Yaskawa INFORM job: R1_W29-KM-NOWY-MP.JBI

/JOB
//NAME R1_W29-KM-NOWY-MP
///FOLDERNAME KRIS-SCIANA
//POS
///NPOS 90,90,76,8,0,0
///TOOL 0
///POSTYPE PULSE
///PULSE
C00000=-43238,-20123,-76298,22793,79190,-61716
C00001=-147206,-71099,-63807,5032,65627,-10001
C00002=-131466,-57276,-50947,-729,64392,-4195
C00003=-131466,-55755,-45239,-747,61662,-4178
C00004=-113506,-33937,-32252,-19801,72986,17092
C00005=-113506,-33758,-31414,-19844,72586,17160
C00006=-113506,-33937,-32252,-19801,72986,17092
C00007=-112868,-36448,-33885,-19979,72871,17349
C00008=-112868,-36201,-32777,-20033,72350,17439
C00009=-113561,-35138,-32088,-19860,72296,17187
C00010=-112868,-36340,-33394,-20002,72641,17389
C00011=-112868,-36673,-34952,-19926,73383,17263
C00012=-136354,-51968,-44201,-1495,62997,-3424
C00013=-136354,-51734,-43329,-1501,62580,-3419
C00014=-136354,-51441,-42272,-1507,62080,-3413
C00015=-136354,-51646,-43010,-1502,62428,-3418
C00016=-136803,-55259,-45028,-1340,61807,-3581
C00017=-136803,-54973,-44058,-1346,61359,-3576
C00018=-136592,-53313,-43138,-1422,61645,-3500
C00019=-136869,-55877,-45678,-1314,61887,-3609
C00020=-144453,-49639,-42868,1535,63375,-6471
C00021=-144614,-48538,-41583,1597,63154,-6534
C00022=-144614,-48258,-40519,1602,62642,-6539
C00023=-144614,-48586,-41775,1593,63247,-6530
C00024=-145217,-51775,-43610,1827,62750,-6765
C00025=-145217,-51364,-42122,1839,62044,-6776
C00026=-144853,-49477,-41036,1695,62343,-6629
C00027=-145217,-51972,-44358,1823,63105,-6759
C00028=-157952,-18054,-25591,12162,79581,-30610
C00029=-158728,-15189,-23240,12317,79720,-30867
C00030=-158728,-15023,-21819,12345,78948,-30943
C00031=-158728,-15162,-22988,12322,79583,-30880
C00032=-160150,-16225,-23788,12608,79748,-31358
C00033=-160150,-16053,-22382,12636,78987,-31435
C00034=-159415,-15465,-21940,12489,78902,-31189
C00035=-160223,-15954,-23704,12620,79843,-31375
C00036=-161879,-22316,-38337,12820,85699,-31343
C00037=-142488,6647,-16194,-2372,99815,22094
C00038=-133363,46346,29890,-18296,105117,75189
C00039=-134257,47901,36105,-18159,102036,75336
C00040=-135288,44692,32242,-18369,102497,74886
C00041=-135288,44939,33433,-18321,101921,74975
C00042=-135288,44745,32503,-18359,102370,74905
C00043=-135129,47566,35532,-18302,102012,75019
C00044=-134852,48227,37162,-18209,101441,75210
C00045=-135455,46185,34960,-18323,101598,74964
C00046=-134852,48227,37162,-18209,101441,75210
C00047=-127142,35074,22200,-17190,105451,77446
C00048=-127142,35126,22513,-17174,105291,77468
C00049=-127142,35298,23490,-17124,104803,77542
C00050=-127142,35126,22513,-17174,105291,77468
C00051=-126238,38948,26146,-16993,105220,77814
C00052=-125881,39159,27623,-16857,104529,78046
C00053=-125732,37116,25510,-16853,104799,78062
C00054=-125881,39159,27623,-16857,104529,78046
C00055=-118491,39693,25202,-15641,107701,80341
C00056=-118491,40027,27191,-15541,106685,80478
C00057=-118491,40312,28701,-15455,105931,80575
C00058=-118491,40115,27679,-15502,106441,80508
C00059=-118523,43718,31472,-15465,105969,80559
C00060=-118523,43964,32657,-15412,105387,80635
C00061=-118326,41786,30355,-15400,105712,80665
C00062=-118523,43964,32657,-15412,105387,80635
C00063=-118101,6095,-16714,-15495,98189,81670
C00064=-121393,-29377,-38195,-9470,79556,5065
C00065=-135587,-47759,-49879,-6114,75955,393
C00066=-135563,-42241,-39607,-6218,72490,575
C00067=-148370,-35238,-35185,1969,72538,-10310
C00068=-156952,-26882,-29550,12128,77113,-24719
C00069=-159766,-12416,-18981,12668,78449,-25578
C00070=-155246,-26379,-37143,3868,78146,-24514
C00071=-111750,-20922,-29619,-16910,84852,24161
C00072=-112985,-19212,-23920,-16796,82079,24108
C00073=-118831,-30060,-31314,-15936,79920,22326
C00074=-124977,-39388,-37559,-9656,73919,11756
C00075=-135123,-42820,-39976,-5392,72032,5771
C00076=-141350,-43617,-40361,1374,71221,-3156
C00077=-141351,-45056,-47095,1351,74625,-3115
C00078=-142962,-17809,-31450,1751,79026,-53612
C00079=-136048,25460,5355,-7693,98061,-70296
C00080=-129481,56377,46609,-18750,110732,-89791
C00081=-130454,29429,16363,-16121,101280,-88696
C00082=-134058,37349,27654,-26404,95753,-89965
C00083=-134055,36228,21042,-26664,98897,-90683
C00084=-119345,38761,21089,-14797,104992,-85146
C00085=-121095,38621,26360,-13285,104325,-87017
C00086=-134151,52750,43450,-11485,107873,-85219
C00087=-130248,33721,13027,-16263,105211,-80194
C00088=-133531,-22452,-45998,-16065,102330,-23096
C00089=-43238,-20123,-76298,22793,79190,-61716
BC00000=125007,760961,1070891
BC00001=266312,761507,1070908
BC00002=266312,761507,1070908
BC00003=266312,761507,1070908
BC00004=266312,761507,1070908
BC00005=266312,761507,1070908
BC00006=266312,761507,1070908
BC00007=266312,761507,1070908
BC00008=266312,761507,1070908
BC00009=266312,761507,1070908
BC00010=266312,761507,1070908
BC00011=266312,761507,1070908
BC00012=266312,761507,1070908
BC00013=266312,761507,1070908
BC00014=266312,761507,1070908
BC00015=266312,761507,1070908
BC00016=266312,761507,1070908
BC00017=266312,761507,1070908
BC00018=266312,761507,1070908
BC00019=266312,761507,1070908
BC00020=266312,761507,1070908
BC00021=266312,761507,1070908
BC00022=266312,761507,1070908
BC00023=266312,761507,1070908
BC00024=266312,761507,1070908
BC00025=266312,761507,1070908
BC00026=266312,761507,1070908
BC00027=266312,761507,1070908
BC00028=266312,761507,1070908
BC00029=266312,761507,1070908
BC00030=266312,761507,1070908
BC00031=266312,761507,1070908
BC00032=266312,761507,1070908
BC00033=266312,761507,1070908
BC00034=266312,761507,1070908
BC00035=266312,761507,1070908
BC00036=266312,761507,1070908
BC00037=266312,761507,1070908
BC00038=266312,761507,1070908
BC00039=266312,761507,1070908
BC00040=266312,761507,1070908
BC00041=266312,761507,1070908
BC00042=266312,761507,1070908
BC00043=266312,761507,1070908
BC00044=266312,761507,1070908
BC00045=266312,761507,1070908
BC00046=266312,761507,1070908
BC00047=266312,761507,1070908
BC00048=266312,761507,1070908
BC00049=266312,761507,1070908
BC00050=266312,761507,1070908
BC00051=266312,761507,1070908
BC00052=266312,761507,1070908
BC00053=266312,761507,1070908
BC00054=266312,761507,1070908
BC00055=266312,761507,1070908
BC00056=266312,761507,1070908
BC00057=266313,761507,1070907
BC00058=266313,761507,1070907
BC00059=266313,761507,1070907
BC00060=266313,761507,1070907
BC00061=266313,761507,1070907
BC00062=266313,761507,1070907
BC00063=266313,761507,1070907
BC00064=266313,761507,1070907
BC00065=266313,761507,1070907
BC00066=266313,761507,1070907
BC00067=266311,761506,1070905
BC00068=266311,761506,1070905
BC00069=266311,761506,1070903
BC00070=266311,761506,1070905
BC00071=266311,761506,1070905
BC00072=266311,761506,1070905
BC00073=266311,761506,1070905
BC00074=266311,761506,1070905
BC00075=266311,761506,1070905
BC00076=266311,761506,1070905
BC00077=266311,761506,1070905
BC00078=266311,761506,1070905
BC00079=270065,761521,1070907
BC00080=274381,761538,1070909
BC00081=274381,761538,1070909
BC00082=274381,761538,1070909
BC00083=274381,761538,1070909
BC00084=274381,761538,1070909
BC00085=274381,761538,1070909
BC00086=274381,761538,1070909
BC00087=274381,761538,1070909
BC00088=274381,761538,1070909
BC00089=125007,760961,1070891
EC00000=-798155,1112952
EC00001=-798156,1112952
EC00002=-798156,1112952
EC00003=-798156,1112952
EC00004=-798156,1112952
EC00005=-798156,1112952
EC00006=-798156,1112952
EC00007=-798156,1112952
EC00008=-798156,1112952
EC00009=-798156,1112952
EC00010=-798156,1112952
EC00011=-798156,1112952
EC00012=-798156,1112952
EC00013=-798156,1112952
EC00014=-798156,1112952
EC00015=-798156,1112952
EC00016=-798156,1112952
EC00017=-798156,1112952
EC00018=-798156,1112952
EC00019=-798156,1112952
EC00020=-798156,1112952
EC00021=-798156,1112952
EC00022=-798156,1112952
EC00023=-798156,1112952
EC00024=-798156,1112952
EC00025=-798156,1112952
EC00026=-798156,1112952
EC00027=-798156,1112952
EC00028=-798156,1112952
EC00029=-798156,1112952
EC00030=-798156,1112952
EC00031=-798156,1112952
EC00032=-798156,1112952
EC00033=-798156,1112952
EC00034=-798156,1112952
EC00035=-798156,1112952
EC00036=-798156,1112952
EC00037=-798156,1112952
EC00038=-798156,1112952
EC00039=-798156,1112952
EC00040=-798156,1112952
EC00041=-798156,1112952
EC00042=-798156,1112952
EC00043=-798156,1112952
EC00044=-798156,1112952
EC00045=-798154,1112952
EC00046=-798154,1112952
EC00047=-798154,1112952
EC00048=-798154,1112952
EC00049=-798154,1112952
EC00050=-798154,1112952
EC00051=-798154,1112952
EC00052=-798154,1112952
EC00053=-798151,1112952
EC00054=-798151,1112952
EC00055=-798147,1112952
EC00056=-798151,1112952
EC00057=-798151,1112952
EC00058=-798151,1112952
EC00059=-798151,1112952
EC00060=-798151,1112952
EC00061=-798151,1112952
EC00062=-798151,1112952
EC00063=-798151,1112952
EC00064=-798151,1112952
EC00065=-798154,1112952
EC00066=-798156,1112952
EC00067=-798156,1112952
EC00068=-798156,1112952
EC00069=-798156,1112952
EC00070=-798156,1112952
EC00071=-798156,1112952
EC00072=-798156,1112952
EC00073=-798156,1112952
EC00074=-798156,1112952
EC00075=-798155,1112952
///POSTYPE BASE
///RECTAN
///RCONF 0,0,0,0,0,0,0,0,0,0,0,0,0,0,0,0,0,0,0,0,0,0,0,0
P00006=0.222,-3.123,-1.508,0.0000,0.0000,0.0000
P00021=-0.225,-6.128,-0.405,0.0000,0.0000,0.0000
P00022=0.222,-3.123,-1.508,0.0000,0.0000,0.0000
P00023=0.143,-0.036,0.682,0.0000,0.0000,0.0000
P00024=0.145,-0.552,1.326,0.0000,0.0000,0.0000
P00025=-2.003,0.006,0.728,0.0000,0.0000,0.0000
P00026=0.562,-0.002,-0.337,0.0000,0.0000,0.0000
P00027=-0.746,0.015,-9.096,0.0000,0.0000,0.0000
//INST
///DATE 2024/07/23 11:59
///ATTR SC,RW
///GROUP1 RB1,BS1
///GROUP2 ST1
NOP
SFTOF
MOVJ C00000 BC00000 VJ=15.00  +MOVJ EC00000 VJ=15.00
MOVJ C00001 BC00001 VJ=50.00  +MOVJ EC00001 VJ=50.00
MOVJ C00002 BC00002 VJ=15.00  +MOVJ EC00002 VJ=15.00
'SEARCH
MOVL C00003 BC00003 V=58.3  +MOVJ EC00003 VJ=15.00
MOVL C00004 BC00004 V=58.3  +MOVJ EC00004 VJ=15.00
REFP 3 RB1 C00005 BC00005
CALL JOB:SEARCH-R1
SET P021 P006
SFTON P021
MOVL C00006 BC00006 V=58.3  +MOVJ EC00005 VJ=15.00
MOVL C00007 BC00007 V=83.3  +MOVJ EC00006 VJ=15.00
MOVL C00008 BC00008 V=83.3  +MOVJ EC00007 VJ=15.00
REFP 3 RB1 C00009 BC00009
CALL JOB:SEARCH-R1
SET P021 P006
SFTON P021
MOVL C00010 BC00010 V=58.3  +MOVJ EC00008 VJ=15.00
MOVL C00011 BC00011 V=100.0  +MOVJ EC00009 VJ=15.00
SFTOF
MOVL C00012 BC00012 V=133.3  +MOVJ EC00010 VJ=15.00
MOVL C00013 BC00013 V=58.3  +MOVJ EC00011 VJ=15.00
REFP 3 RB1 C00014 BC00014
CALL JOB:SEARCH-R1
SET P022 P006
SFTON P022
MOVL C00015 BC00015 V=58.3  +MOVJ EC00012 VJ=15.00
MOVL C00016 BC00016 V=100.0  +MOVJ EC00013 VJ=15.00
MOVL C00017 BC00017 V=100.0  +MOVJ EC00014 VJ=15.00
REFP 3 RB1 C00018 BC00018
CALL JOB:SEARCH-R1
SET P022 P006
SFTON P022
MOVL C00019 BC00019 V=100.0  +MOVJ EC00015 VJ=15.00
SFTOF
MOVL C00020 BC00020 V=166.7  +MOVJ EC00016 VJ=15.00
MOVL C00021 BC00021 V=58.3  +MOVJ EC00017 VJ=15.00
REFP 3 RB1 C00022 BC00022
CALL JOB:SEARCH-R1
SET P023 P006
SFTON P023
MOVL C00023 BC00023 V=58.3  +MOVJ EC00018 VJ=15.00
MOVL C00024 BC00024 V=83.3  +MOVJ EC00019 VJ=15.00
MOVL C00025 BC00025 V=83.3  +MOVJ EC00020 VJ=15.00
REFP 3 RB1 C00026 BC00026
CALL JOB:SEARCH-R1
SET P023 P006
SFTON P023
MOVL C00027 BC00027 V=100.0  +MOVJ EC00021 VJ=15.00
MOVL C00028 BC00028 V=100.0  +MOVJ EC00022 VJ=15.00
SFTOF
MOVL C00029 BC00029 V=58.3  +MOVJ EC00023 VJ=15.00
REFP 3 RB1 C00030 BC00030
CALL JOB:SEARCH-R1
SET P024 P006
SFTON P024
MOVL C00031 BC00031 V=58.3  +MOVJ EC00024 VJ=15.00
MOVL C00032 BC00032 V=100.0  +MOVJ EC00025 VJ=15.00
MOVL C00033 BC00033 V=100.0  +MOVJ EC00026 VJ=15.00
REFP 3 RB1 C00034 BC00034
CALL JOB:SEARCH-R1
SET P024 P006
SFTON P024
MOVL C00035 BC00035 V=100.0  +MOVJ EC00027 VJ=15.00
SSFTOF
MOVJ C00036 BC00036 VJ=100.00  +MOVJ EC00028 VJ=100.00
MOVJ C00037 BC00037 VJ=100.00  +MOVJ EC00029 VJ=100.00
MOVJ C00038 BC00038 VJ=100.00  +MOVJ EC00030 VJ=100.00
MOVL C00039 BC00039 V=166.7  +MOVJ EC00031 VJ=15.00
MOVL C00040 BC00040 V=58.3  +MOVJ EC00032 VJ=15.00
REFP 3 RB1 C00041 BC00041
CALL JOB:SEARCH-R1
SET P025 P006
SFTON P025
MOVL C00042 BC00042 V=58.3  +MOVJ EC00033 VJ=15.00
MOVL C00043 BC00043 V=100.0  +MOVJ EC00034 VJ=15.00
MOVL C00044 BC00044 V=100.0  +MOVJ EC00035 VJ=15.00
REFP 3 RB1 C00045 BC00045
CALL JOB:SEARCH-R1
SET P025 P006
SFTON P025
MOVL C00046 BC00046 V=100.0  +MOVJ EC00036 VJ=15.00
SSFTOF
MOVL C00047 BC00047 V=250.0  +MOVJ EC00037 VJ=100.00
MOVL C00048 BC00048 V=58.3  +MOVJ EC00038 VJ=15.00
REFP 3 RB1 C00049 BC00049
CALL JOB:SEARCH-R1
SET P026 P006
SFTON P026
MOVL C00050 BC00050 V=58.3  +MOVJ EC00039 VJ=15.00
MOVL C00051 BC00051 V=100.0  +MOVJ EC00040 VJ=15.00
MOVL C00052 BC00052 V=100.0  +MOVJ EC00041 VJ=15.00
REFP 3 RB1 C00053 BC00053
CALL JOB:SEARCH-R1
SET P026 P006
SFTON P026
MOVL C00054 BC00054 V=100.0  +MOVJ EC00042 VJ=15.00
MOVL C00055 BC00055 V=250.0  +MOVJ EC00043 VJ=100.00
MOVL C00056 BC00056 V=58.3  +MOVJ EC00044 VJ=15.00
REFP 3 RB1 C00057 BC00057
CALL JOB:SEARCH-R1
SET P027 P006
SFTON P027
MOVL C00058 BC00058 V=58.3  +MOVJ EC00045 VJ=15.00
MOVL C00059 BC00059 V=100.0  +MOVJ EC00046 VJ=15.00
MOVL C00060 BC00060 V=100.0  +MOVJ EC00047 VJ=15.00
REFP 3 RB1 C00061 BC00061
CALL JOB:SEARCH-R1
SET P027 P006
SFTON P027
MOVL C00062 BC00062 V=100.0  +MOVJ EC00048 VJ=15.00
SFTOF
MOVJ C00063 BC00063 VJ=100.00  +MOVJ EC00049 VJ=100.00
MOVJ C00064 BC00064 VJ=100.00  +MOVJ EC00050 VJ=100.00
MOVJ C00065 BC00065 VJ=100.00  +MOVJ EC00051 VJ=100.00
SFTON P023
MOVL C00066 BC00066 V=100.0 PL=0  +MOVJ EC00052 VJ=15.00
MACRO1 MJ#(0) ARGF7
ARCON
MOVL C00067 BC00067 V=10.8  +MOVJ EC00053 VJ=15.00
MOVL C00068 BC00068 V=10.8  +MOVJ EC00054 VJ=15.00
SFTON P024
MOVL C00069 BC00069 V=10.8  +MOVJ EC00055 VJ=15.00
ARCOF
SFTOF
MOVJ C00070 BC00070 VJ=30.00  +MOVJ EC00056 VJ=15.00
MOVJ C00071 BC00071 VJ=100.00  +MOVJ EC00057 VJ=100.00
SFTOF
SFTON P021
MOVL C00072 BC00072 V=100.0 PL=0  +MOVJ EC00058 VJ=15.00
ARCON
MOVL C00073 BC00073 V=10.8  +MOVJ EC00059 VJ=15.00
MOVL C00074 BC00074 V=10.8  +MOVJ EC00060 VJ=15.00
SFTON P022
MOVL C00075 BC00075 V=10.8  +MOVJ EC00061 VJ=15.00
MOVL C00076 BC00076 V=10.8  +MOVJ EC00062 VJ=15.00
ARCOF
MOVJ C00077 BC00077 VJ=15.00  +MOVJ EC00063 VJ=15.00
SFTOF
MOVJ C00078 BC00078 VJ=100.00  +MOVJ EC00064 VJ=100.00
MOVJ C00079 BC00079 VJ=100.00  +MOVJ EC00065 VJ=100.00
MOVJ C00080 BC00080 VJ=50.00  +MOVJ EC00066 VJ=50.00
SFTOF
SFTON P026
MOVL C00081 BC00081 V=250.0 PL=0  +MOVJ EC00067 VJ=15.00
ARCON
SFTON P025
MOVL C00082 BC00082 V=10.8  +MOVJ EC00068 VJ=15.00
ARCOF
MOVJ C00083 BC00083 VJ=15.00  +MOVJ EC00069 VJ=15.00
SFTOF
MOVJ C00084 BC00084 VJ=15.00  +MOVJ EC00070 VJ=15.00
SFTON P027
MOVL C00085 BC00085 V=100.0 PL=0  +MOVJ EC00071 VJ=15.00
ARCON
SFTON P026
MOVL C00086 BC00086 V=10.8  +MOVJ EC00072 VJ=15.00
ARCOF
SFTOF
MOVJ C00087 BC00087 VJ=15.00  +MOVJ EC00073 VJ=15.00
MOVJ C00088 BC00088 VJ=100.00  +MOVJ EC00074 VJ=100.00
MOVJ C00089 BC00089 VJ=100.00  +MOVJ EC00075 VJ=20.00
SFTOF
END
